FUNCTION_BLOCK PUBLIC Motors
VAR_INPUT
	ACPosition: INT;
	CurrentPosition: INT;
	Movement: BOOL;
	Direction: BOOL;
END_VAR
VAR_OUTPUT
END_VAR
VAR
END_VAR

END_FUNCTION_BLOCK

(* stored: Version 1.1.0.1, ProductVersion 3.1.4024.13
   POU Motors: Id {a60a75ec-7bee-40de-97f9-a42bfc7b267c}, SpecialFunc None *)
